(* task info with times of current task converted to millisecs and microsecs *)
FUNCTION_BLOCK FB_SYSTEM_TaskInfo
VAR_INPUT
END_VAR
VAR_OUTPUT
	stPLCTaskSys		:	PlcTaskSystemInfo;
	tTaskTimeMillisecs	: TIME;		(* Task Time in time format with ms resolution *)
	fTaskTimeMicrosecs	: LREAL;	(* Task Time in LREAL format with us resolution *)
	nTaskIndex			: BYTE;		(* Task Index of task where this FB is called *)
END_VAR
VAR	
	fbGetCurTaskIdx 				: 	GETCURTASKINDEX;
END_VAR
(*
-------------------------------------------------------------------------------------------------
Date		Version	Author	Comments
-------------------------------------------------------------------------------------------------
30/01/2015	3.00.00	PB		No change

-------------------------------------------------------------------------------------------------
15/03/2010	1.01.00	PB		Current PLC Port No added to FB_TaskTime
							bFirstCycle made primary output of FB_TaskTime
05/02/2010	1.00.00	PB		Initial release
							
-------------------------------------------------------------------------------------------------
*)

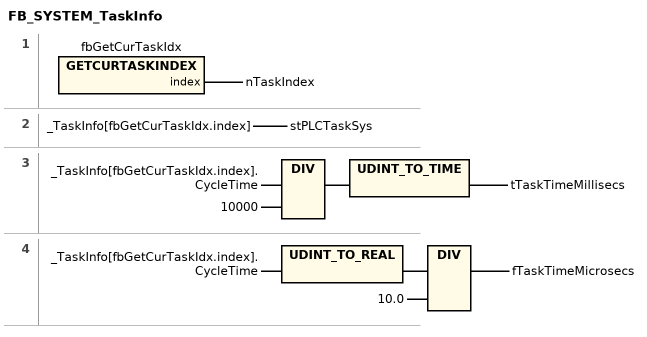
// NETWORK 1
fbGetCurTaskIdx(); // GETCURTASKINDEX
nTaskIndex := fbGetCurTaskIdx.index;

// NETWORK 2
stPLCTaskSys := _TaskInfo[fbGetCurTaskIdx.index];

// NETWORK 3
tTaskTimeMillisecs := UDINT_TO_TIME(_TaskInfo[fbGetCurTaskIdx.index].CycleTime / 10000);

// NETWORK 4
fTaskTimeMicrosecs := UDINT_TO_REAL(_TaskInfo[fbGetCurTaskIdx.index].CycleTime) / 10.0;

END_FUNCTION_BLOCK

(* stored: Version 1.1.0.1
   POU FB_SYSTEM_TaskInfo: Id {7f4e8961-2816-45e6-9ab8-3663e1a3d672}, SpecialFunc None *)
